// TIA Portal V16 export
// export: Created 2021-04-11T09:51:32.5827485Z, ExportSetting WithDefaults, DisplayName Totally Integrated Automation Portal, DisplayVersion V16, DisplayName TIA Portal Version Control Interface, DisplayVersion V16, DisplayName TIA Portal Openness, DisplayVersion V16, DisplayName STEP 7 Professional, DisplayVersion V16, DisplayName STEP 7 Safety, DisplayVersion V16, DisplayName WinCC Unified SCADA Engineering System, DisplayVersion V16
FUNCTION "bitMaskSortFor" : Void   // FC6, LAD
{ S7_Optimized_Access := 'TRUE' }
VERSION : 0.1
// stored: AutoNumber true, IsIECCheckEnabled false, SetENOAutomatically false, UDAEnableTagReadback false
   VAR_INPUT
      value : DInt;
   END_VAR
   VAR_IN_OUT
      bitMask : Array[0..12] of Bool;
   END_VAR
BEGIN

REGION Network 1 (SCL)
   #bitMask[0] := #value.%X0;
   #bitMask[1] := #value.%X1;
   #bitMask[2] := #value.%X2;
   #bitMask[3] := #value.%X3;
   #bitMask[4] := #value.%X4;
   #bitMask[5] := #value.%X5;
   #bitMask[6] := #value.%X6;
   #bitMask[7] := #value.%X7;
   #bitMask[8] := #value.%X8;
   #bitMask[9] := #value.%X9;
   #bitMask[10] := #value.%X10;
   #bitMask[11] := #value.%X11;
   #bitMask[12] := #value.%X12;
END_REGION
END_FUNCTION
